DEVICE_TYPE _CB_TCREST
  (* Standard: 61499-2 *)
  (* Version 0.1, 2019-00-29, hpea485, UOA *)
  RESOURCE Resource : _CBCore0
  END_RESOURCE
  RESOURCE Resource1 : _CBCore1
  END_RESOURCE
  RESOURCE Resource2 : _CBCore2
  END_RESOURCE
  RESOURCE Resource3 : _CBCore3
  END_RESOURCE
END_DEVICE_TYPE
